TYPE Cnv_Inputs_DUT :
STRUCT
	Forward_Sensor:	BOOL;
	Backward_Sensor:	BOOL;
	VFD_Status:	WORD;
	VFD_Speed_Actual:	INT;
	VFD_ActualCurrent:	INT;
	VFD_ActualTorque:	INT;
END_STRUCT
END_TYPE

(* stored: Version 1.1.0.1
   DUT Cnv_Inputs_DUT: Id {f19e415e-bf3c-45c0-bc8d-2543a824b9d0} *)
